{attribute 'qualified_only'}
{attribute 'strict'}
{attribute 'to_string'}
TYPE E_UnitError :
(
    None,
    SafetyNotOk,
    NotHomed,
    Timeout,
    VacuumNotOk,
    SensorFault
);
END_TYPE

(* stored: Version 1.1.0.1
   DUT E_UnitError: Id {60b25982-15ad-4444-ba52-73a7af784509} *)
